// TIA Portal project "Project1" (V15)

(* hardware
DEVICE "S7-1200 station_1"  S7-1200 Station
   slot 0: "Rack_0"  S7-1200 Rack  Rack  V1.0
   slot 1: "PLC_1"  CPU 1214C DC/DC/Rly  6ES7 214-1HG40-0XB0  V4.2
*)

// ===== PLC "PLC_1"  CPU 1214C DC/DC/Rly =====

VAR_GLOBAL   // PLC tag table "Default tag table"
   ""qXiloRice1"" AT %Q0.0 : Bool;
   ""qXiloRice2"" AT %Q0.1 : Bool;
   ""qXiloRice3"" AT %Q0.2 : Bool;
   ""qXiloCorn4"" AT %Q0.3 : Bool;
   ""qXiloCorn5"" AT %Q0.4 : Bool;
   ""qXiloCorn6"" AT %Q0.5 : Bool;
   ""qXiloCorn7"" AT %Q0.6 : Bool;
   ""qXiloCassava8"" AT %Q0.7 : Bool;
   ""qXiloCassava9"" AT %Q1.0 : Bool;
   ""qXiloBean10"" AT %Q1.1 : Bool;
   ""qXiloBean11"" AT %Q1.2 : Bool;
   ""qXiloBean12"" AT %Q1.3 : Bool;
   ""qXiloFish13"" AT %Q1.4 : Bool;
   ""qXiloFish14"" AT %Q1.5 : Bool;
   ""qXiloFish15"" AT %Q1.6 : Bool;
   ""qXiloFish16"" AT %Q1.7 : Bool;
   ""qValveScale1"" AT %Q2.0 : Bool;
   ""qValveScale2"" AT %Q2.1 : Bool;
   ""qMotorMixTank"" AT %Q2.2 : Bool;
   ""qValveMixTank"" AT %Q2.3 : Bool;
END_VAR